# EPICS autosave request: dxp/tags/R2-4/iocBoot/iocSaturn/auto_settings_med.req
file "simple_mca_settings.req",  P=dxpSaturn:med:, M=mca1
file "dxp_settings.req",         P=dxpSaturn:med:, R=dxp1
